RoboDK station: conveyor.rdk

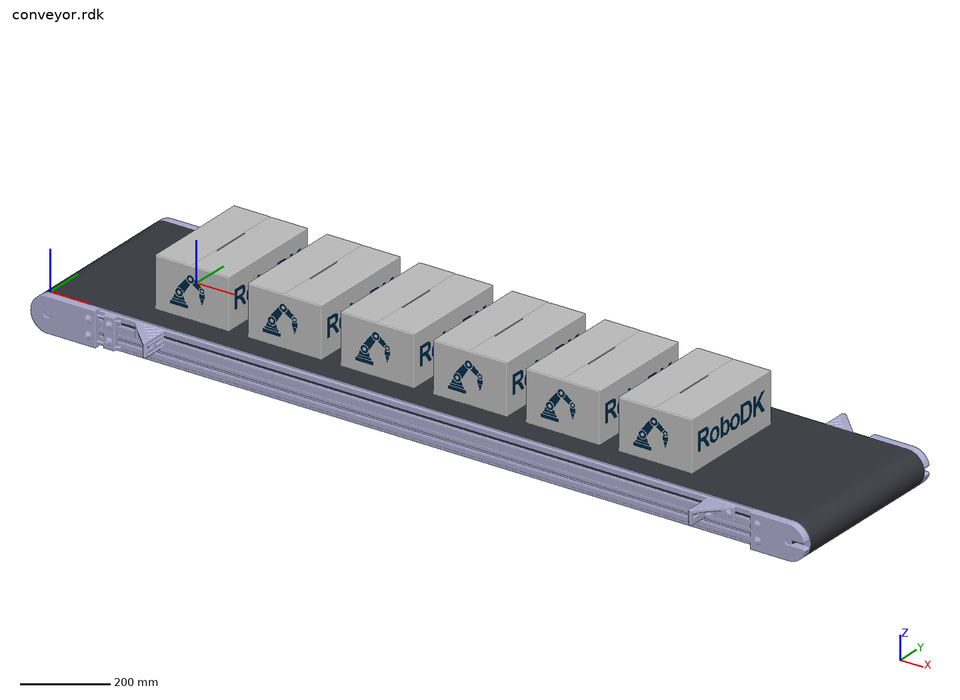
[picture v0: the station drawn from its stored meshes, robots at their saved joint values, targets as dots, program paths as lines]
Station conveyor (saved by RoboDK 5.9.2). Poses are relative to the parent item; angles as X-Y-Z fixed-axis rotations.
  - frame Conveyor Belt (2m) Base at (0, 0, 0) mm
    - robot Conveyor Belt (2m): 1 axes
        modified DH rows (alpha deg, a mm, theta deg, d mm): 0, 0, 0, 0 linear
        base shift (0, 0, 0) mm, rotated rx 0 ry 90 rz 0 deg
        joint limits [-500000] to [500000]; home [0]; saved at [240]
      - frame Frame 2 at (0, 220, 0) mm
        - object Box 1 at (0, -160, 0) mm, size 199 x 305.1 x 133.7 mm, geometry from Box-12x7in-Closed.sld
        - object Box 2 at (250, -160, 0) mm, size 199 x 305.1 x 133.7 mm, geometry from Box-12x7in-Closed.sld
        - object Box3 at (500, -160, 0) mm, size 199 x 305.1 x 133.7 mm, geometry from Box-12x7in-Closed.sld
        - object Box 4 at (750, -160, 0) mm, size 199 x 305.1 x 133.7 mm, geometry from Box-12x7in-Closed.sld
        - object Box 5 at (1000, -160, 0) mm, size 199 x 305.1 x 133.7 mm, geometry from Box-12x7in-Closed.sld
        - object Box 6 at (1250, -160, 0) mm, size 199 x 305.1 x 133.7 mm, geometry from Box-12x7in-Closed.sld
  - Python program InitConveyor (listed below)
  - Python program Conveyor Next Part (listed below)

--- Python program InitConveyor ---
# Forward and backwards compatible use of the RoboDK API:
# Remove these 2 lines to follow python programming guidelines
from robodk import *      # RoboDK API
from robolink import *    # Robot toolbox
# Link to RoboDK
RDK = Robolink()

CONVEYOR ='Conveyor Belt'
mechanism = RDK.Item(CONVEYOR, itemtype=ITEM_TYPE_ROBOT)


if mechanism.Valid():
    mechanism.setJoints([0])

--- Python program Conveyor Next Part ---
# Type help("robodk.robolink") or help("robodk.robomath") for more information
# Press F5 to run the script
# Documentation: https://robodk.com/doc/en/RoboDK-API.html
# Reference:     https://robodk.com/doc/en/PythonAPI/robodk.html
# Note: It is not required to keep a copy of this file, your Python script is saved with your RDK project

# Forward and backwards compatible use of the RoboDK API:
# Remove these 2 lines to follow python programming guidelines
from robodk import *      # RoboDK API
from robolink import *    # Robot toolbox
# Link to RoboDK
RDK = Robolink()

CONVEYOR = 'Conveyor Belt'
mechanism = RDK.Item(CONVEYOR, itemtype= ITEM_TYPE_ROBOT)

PART_TRAVEL_MM = -300
if mechanism.Valid():
    mechanism.MoveJ(mechanism.Joints() + PART_TRAVEL_MM)
